# EPICS StreamDevice protocol: sdgEliteApp/Db/sdgEliteV1.proto
# Use this file if the "Set newline to host" option (set:ser:nl) has been set.

# This device can mix up send/receive strings.  Using the @mismatch handlers fixes it.
# Fixed 12/8/16 md

InTerminator = "Ok\r\n";
OutTerminator = "\r";

stausMismatch = "status?\r";

#ReadTimeout = 10000;
#LockTimeout = 10000;
#ReplyTimeout = 10000;
#WriteTimeout = 3000;

getStatus {
    Separator=",";
    out "status?";
    in "%s";
    @mismatch {
    in "Ok\r\n";
    }
}

getBWDDiodeStat {
    out "read:sta:bwd?";
    in "%{0|1}";
    @mismatch {
    in $stausMismatch;
    }
}

getBWDIntStat {
    out "read:bwd?";
    in "%{0|1}";
    @mismatch {
    in $stausMismatch;
    }
}

resetBWD {
    out "reset";
    in "";
    @mismatch {
    in $stausMismatch;
    }
}

setBWDThresh {
    out "set:bwd:lv %i";
    in "";
    @mismatch {
    in $stausMismatch;
    }
}

getCh {
    out "read:c\$1?";
    in "%d,%*d\r\n";
    @mismatch {
    in $stausMismatch;
    }
}

setCh {
    out "set:c\$1 %{0|1}";
    in "";
    @mismatch {
    in $stausMismatch;
    }
}

getDelay {
    out "read:del:c\$1?";
    in "%f\r\n";
    @mismatch {
    in $stausMismatch;
    }
}

setDelay {
    out "set:del:c\$1 %.2f";
    in "";
    @mismatch {
    in $stausMismatch;
    }
}
